(* CODESYS project BagFeedMotor_.xml

Project tree, tasks and I/O mapping:
  function block BagFeedMotor_ [CFC]
*)

// BagFeedMotor_
FUNCTION_BLOCK BagFeedMotor_
VAR_INPUT
	ExecuteMove: 		BOOL; 				// Execute a step and direction incremental move
	Direction: 			UINT; 				// 1 = Forward, 0 = Reverse
	Steps: 				UDINT := 3000; 		// Number of motor pulses for incremental move
	Speed: 				UINT;				// Speed 
	TriggerOnSensor: 	BOOL;				//
	JogForward: 		BOOL;				// 
	JogReverse: 		BOOL;				// 
	Count: 				UDINT;				// Current Count
	Rate: 				UDINT; 				// Current Rate
	ResetCount: 		BOOL;				// Reset pulse count
	Settings: 			BagFeedMotorSettings;
	MaxSpeed: 			UINT := 2000;		//
	LabelSensor: 		BOOL;				//
END_VAR
VAR_OUTPUT
	Forward: 			BOOL;				// Move forward
	Reverse: 			BOOL;				// Move reverse
	ResetAlarmOutput: 	BOOL;				// Reset alarm output to motor controller
	SpeedOutput: 		UINT;				// Analog speed output to motor controller
	Complete: 			BOOL;				// Pulses TRUE when a move command has completed 
	InputFunction: 		UINT;				// High speed counter setting, 1 = Simple Count
	CounterLimit: 		UDINT;				// High speed counter maximum count
	RateChannel: 		UINT;				// High speed counter window = 1
	RateTime: 			UINT;				// High speed counter rate time in milliseconds = 1000
	CounterCommand: 	UINT;				// High speed counter command 0 = Keep Counting, 1 = Stop Counting, 2 = Clear Count
END_VAR
VAR
	_ManualJogForward: 	BOOL;
	_ManualJogReverse: 	BOOL;
	_ManualResetCount: 	BOOL;
	_MoveFunction: 		BagFeedMotorIMove;
	_ManualStopMotor: 	BOOL;
	//_CompleteTimer: 	TOF;
	_ExecuteTrigger: 	R_TRIG;
	_PID_0: 			PID;
	//_KP: 				REAL;
	//_KI: 				REAL;
	//_KD: 				REAL;
	//_Y_MIN: 			REAL;
	//_Y_MAX: 			REAL;
	StaticSpeed: 		BOOL;
	_LabelTrigger: 		F_TRIG;
END_VAR
VAR // added by the converter: edge detectors and wires of the graphical bodies
    _w1, _w3 : BOOL;
    _w2 : UINT;
    _w4 : ANY;
END_VAR

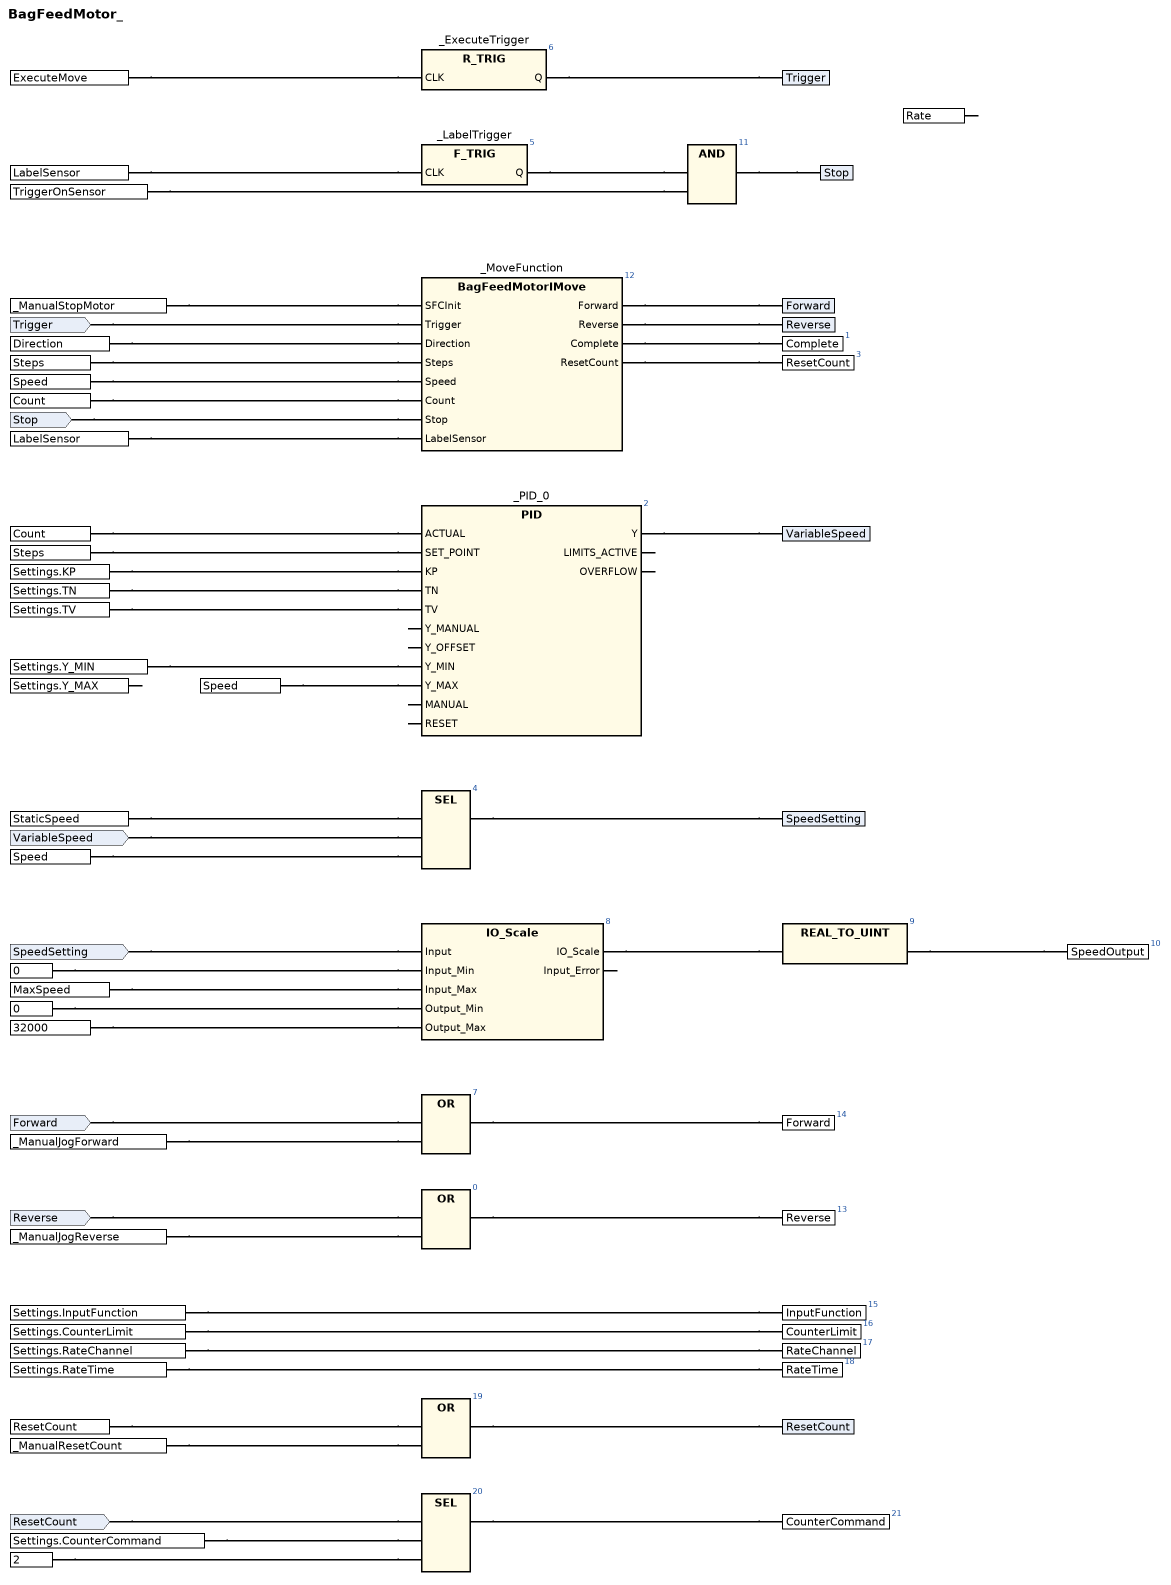
_w1 := _MoveFunction.Reverse OR _ManualJogReverse;
Complete := _MoveFunction.Complete;
_PID_0(
    ACTUAL := Count,
    SET_POINT := Steps,
    KP := Settings.KP,
    TN := Settings.TN,
    TV := Settings.TV,
    Y_MIN := Settings.Y_MIN,
    Y_MAX := Speed); // PID
ResetCount := _MoveFunction.ResetCount;
_w2 := SEL(StaticSpeed, _PID_0.Y, Speed);
_LabelTrigger(CLK := LabelSensor); // F_TRIG
_ExecuteTrigger(CLK := ExecuteMove); // R_TRIG
_w3 := _MoveFunction.Forward OR _ManualJogForward;
_w4 := IO_Scale(Input := _w2, Input_Min := 0, Input_Max := MaxSpeed, Output_Min := 0, Output_Max := 32000);
SpeedOutput := REAL_TO_UINT(_w4);
_MoveFunction(
    SFCInit := _ManualStopMotor,
    Trigger := _ExecuteTrigger.Q,
    Direction := Direction,
    Steps := Steps,
    Speed := Speed,
    Count := Count,
    Stop := _LabelTrigger.Q AND TriggerOnSensor,
    LabelSensor := LabelSensor); // BagFeedMotorIMove
Reverse := _w1;
Forward := _w3;
InputFunction := Settings.InputFunction;
CounterLimit := Settings.CounterLimit;
RateChannel := Settings.RateChannel;
RateTime := Settings.RateTime;
CounterCommand := SEL(ResetCount OR _ManualResetCount, Settings.CounterCommand, 2);
// Rate: input not connected
// Settings.Y_MAX: input not connected

END_FUNCTION_BLOCK
